// TIA Portal project "modbus" (V14)

(* hardware
DEVICE "S7-1200 station_1"  S7-1200 Station
   slot 0: "Rack_0"  S7-1200 Rack  Rack  V1.0
   slot 1: "PLC_1"  CPU 1215C DC/DC/DC  6ES7 215-1AG40-0XB0  V4.2
*)

// ===== PLC "PLC_1"  CPU 1215C DC/DC/DC =====

VAR_GLOBAL   // PLC tag table "Default tag table"
   "System_Byte" AT %MB1 : Byte;
   "FirstScan" AT %M1.0 : Bool;
   "DiagStatusUpdate" AT %M1.1 : Bool;
   "AlwaysTRUE" AT %M1.2 : Bool;
   "AlwaysFALSE" AT %M1.3 : Bool;
   "Clock_Byte" AT %MB0 : Byte;
   "Clock_10Hz" AT %M0.0 : Bool;
   "Clock_5Hz" AT %M0.1 : Bool;
   "Clock_2.5Hz" AT %M0.2 : Bool;
   "Clock_2Hz" AT %M0.3 : Bool;
   "Clock_1.25Hz" AT %M0.4 : Bool;
   "Clock_1Hz" AT %M0.5 : Bool;
   "Clock_0.625Hz" AT %M0.6 : Bool;
   "Clock_0.5Hz" AT %M0.7 : Bool;
END_VAR

DATA_BLOCK "DB_ModbusTCP_Connect"   // DB10
{ S7_Optimized_Access := 'TRUE' }
VERSION : 0.1
   VAR
      MBTCPClientRead : TCON_IP_v4;
      MBTCPClientRead_DISCONNECT : Bool;
      MBTCPClientRead_BUSY : Bool;
      MBTCPClientRead_ERROR : Bool;
      MBTCPClientRead_STATUS : Word;
   END_VAR
BEGIN
   MBTCPClientRead.InterfaceId := 64;
   MBTCPClientRead.ID := 16#1;
   MBTCPClientRead.ActiveEstablished := 1;
   MBTCPClientRead.RemoteAddress.ADDR[1] := 16#C0;
   MBTCPClientRead.RemoteAddress.ADDR[2] := 16#A8;
   MBTCPClientRead.RemoteAddress.ADDR[4] := 16#64;
   MBTCPClientRead.RemotePort := 502;
   MBTCPClientRead.LocalPort := 502;
END_DATA_BLOCK

DATA_BLOCK "MBTCP_read_Data"   // DB11
{ S7_Optimized_Access := 'FALSE' }
VERSION : 0.1
   VAR
      Read : Array[1..120] of Word;
   END_VAR
BEGIN
END_DATA_BLOCK

FUNCTION "FC_MBTCP_Client" : Void   // FC10, LAD
{ S7_Optimized_Access := 'TRUE' }
VERSION : 0.1
BEGIN

REGION Network 1
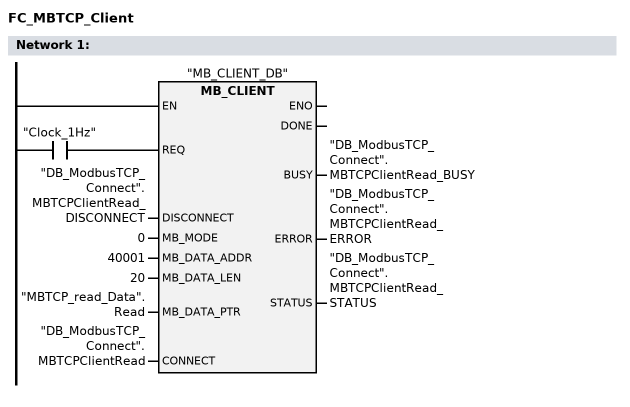
   "MB_CLIENT_DB"(REQ := "Clock_1Hz",   // MB_CLIENT
                  DISCONNECT := "DB_ModbusTCP_Connect".MBTCPClientRead_DISCONNECT,
                  MB_MODE := 0,
                  MB_DATA_ADDR := 40001,
                  MB_DATA_LEN := 20,
                  MB_DATA_PTR := "MBTCP_read_Data".Read,
                  CONNECT := "DB_ModbusTCP_Connect".MBTCPClientRead,
                  BUSY => "DB_ModbusTCP_Connect".MBTCPClientRead_BUSY,
                  ERROR => "DB_ModbusTCP_Connect".MBTCPClientRead_ERROR,
                  STATUS => "DB_ModbusTCP_Connect".MBTCPClientRead_STATUS);
END_REGION
END_FUNCTION

ORGANIZATION_BLOCK "Main"   // OB1, LAD, ProgramCycle
TITLE = "Main Program Sweep (Cycle)"
{ S7_Optimized_Access := 'TRUE' }
VERSION : 0.1
   VAR_INPUT
      Initial_Call : Bool;   // Initial call of this OB
      Remanence : Bool;   // =True, if remanent data are available
   END_VAR
BEGIN

REGION Network 1
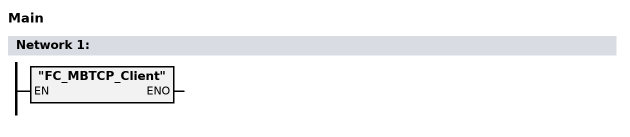
   RUNG wire#powerrail
      "FC_MBTCP_Client"()
   END_RUNG
   // the same network as SCL:
   "FC_MBTCP_Client"();
END_REGION
END_ORGANIZATION_BLOCK